TYPE Conveyor :
STRUCT
	//start : BOOL;
	is_started :  BOOL;
	status : INT;
	id : INT;
    red_light_on : BOOL;
    yellow_light_on : BOOL;
    green_light_on : BOOL;
    in_sensor : BOOL;
    out_sensor : BOOL;
    motor_on : BOOL;
	stop : BOOL;
//	was_stopped : BOOL;
	test_lights : BOOL;
END_STRUCT
END_TYPE

(* stored: Version 1.1.0.1
   DUT Conveyor: Id {2f4ed8bc-eda6-431d-9129-60af6c5a411c} *)
